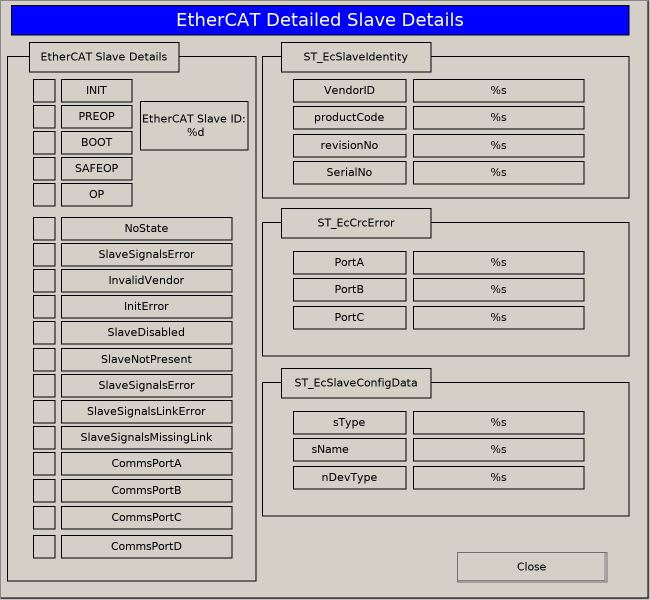
VISUALIZATION diagEtherCATSlaveDetail  // 650x600
VAR_IN_OUT
	//DetailedDataValues:typeEtherCATIndicator;
END_VAR
    Rectangle (0,0 648x598)
    Rectangle (262,56 367x142)
    Rectangle (7,56 249x525)
    Rectangle (33,79 22x23), colour toggle: etherCATdiag.detailDiag.currentState.state = EtherCATstate.INIT
    Rectangle (61,79 71x23), "INIT"
    Rectangle (33,105 22x23), colour toggle: etherCATdiag.detailDiag.currentState.state = EtherCATstate.PREOP
    Rectangle (61,105 71x23), "PREOP"
    Rectangle (33,131 22x23), colour toggle: etherCATdiag.detailDiag.currentState.state = EtherCATstate.BOOT
    Rectangle (61,131 71x23), "BOOT"
    Rectangle (33,157 22x23), colour toggle: etherCATdiag.detailDiag.currentState.state = EtherCATstate.SAFEOP
    Rectangle (61,157 71x23), "SAFEOP"
    Rectangle (33,183 22x23), colour toggle: etherCATdiag.detailDiag.currentState.state = EtherCATstate.OP
    Rectangle (61,183 71x23), "OP"
    Rectangle (33,217 22x23), colour toggle: etherCATdiag.detailDiag.currentState.suffix = EtherCATSuffix.NoState
    Rectangle (61,217 171x23), "NoState"
    Rectangle (33,243 22x23), colour toggle: etherCATdiag.detailDiag.currentState.suffix = EtherCATSuffix.SlaveSignalsError
    Rectangle (61,243 171x23), "SlaveSignalsError"
    Rectangle (33,269 22x23), colour toggle: etherCATdiag.detailDiag.currentState.suffix = EtherCATSuffix.InvalidVendor
    Rectangle (61,269 171x23), "InvalidVendor"
    Rectangle (33,295 22x23), colour toggle: etherCATdiag.detailDiag.currentState.suffix = EtherCATSuffix.InitError
    Rectangle (61,295 171x23), "InitError"
    Rectangle (33,321 22x23), colour toggle: etherCATdiag.detailDiag.currentState.suffix = EtherCATSuffix.SlaveDisabled
    Rectangle (61,321 171x23), "SlaveDisabled"
    Rectangle (33,348 22x23), colour toggle: etherCATdiag.detailDiag.currentState.suffix = EtherCATSuffix.SlaveNotPresent
    Rectangle (61,348 171x23), "SlaveNotPresent"
    Rectangle (33,374 22x23), colour toggle: etherCATdiag.detailDiag.currentState.suffix = EtherCATSuffix.SlaveSignalsError
    Rectangle (61,374 171x23), "SlaveSignalsError"
    Rectangle (33,400 22x23), colour toggle: etherCATdiag.detailDiag.currentState.suffix = EtherCATSuffix.SlaveSignalsLinkError
    Rectangle (61,400 171x23), "SlaveSignalsLinkError"
    Rectangle (33,426 22x23), colour toggle: etherCATdiag.detailDiag.currentState.suffix = EtherCATSuffix.SlaveSignalsMissingLink
    Rectangle (61,426 171x23), "SlaveSignalsMissingLink"
    Rectangle (33,452 22x23), colour toggle: etherCATdiag.detailDiag.currentState.suffix = EtherCATSuffix.CommsPortA
    Rectangle (61,452 171x23), "CommsPortA"
    Rectangle (33,479 22x23), colour toggle: etherCATdiag.detailDiag.currentState.suffix = EtherCATSuffix.CommsPortB
    Rectangle (61,479 171x23), "CommsPortB"
    Rectangle (33,506 22x23), colour toggle: etherCATdiag.detailDiag.currentState.suffix = EtherCATSuffix.CommsPortC
    Rectangle (61,506 171x23), "CommsPortC"
    Rectangle (33,535 22x23), colour toggle: etherCATdiag.detailDiag.currentState.suffix = EtherCATSuffix.CommsPortD
    Rectangle (61,535 171x23), "CommsPortD"
    Rectangle (29,42 150x30), "EtherCAT Slave Details"
    Rectangle (293,79 113x23), "VendorID"
    Rectangle (413,79 171x23), "%s", text variable: etherCATdiag.detailDiag.ConfigData.stSlaveIdentity.vendorId
    Rectangle (413,106 171x23), "%s", text variable: etherCATdiag.detailDiag.ConfigData.stSlaveIdentity.productCode
    Rectangle (293,106 113x23), "productCode"
    Rectangle (293,134 113x23), "revisionNo"
    Rectangle (413,134 171x23), "%s", text variable: etherCATdiag.detailDiag.ConfigData.stSlaveIdentity.revisionNo
    Rectangle (413,161 171x23), "%s", text variable: etherCATdiag.detailDiag.ConfigData.stSlaveIdentity.serialNo
    Rectangle (293,161 113x23), "SerialNo"
    Rectangle (281,42 150x30), "ST_EcSlaveIdentity"
    Rectangle (262,222 367x134)
    Rectangle (293,251 113x23), "PortA"
    Rectangle (413,251 171x23), "%s", text variable: etherCATdiag.detailDiag.crcCount.portA
    Rectangle (413,278 171x23), "%s", text variable: etherCATdiag.detailDiag.crcCount.portB
    Rectangle (293,278 113x23), "PortB"
    Rectangle (293,306 113x23), "PortC"
    Rectangle (413,306 171x23), "%s", text variable: etherCATdiag.detailDiag.crcCount.portC
    Rectangle (281,208 150x30), "ST_EcCrcError"
    Rectangle (262,382 367x134)
    Rectangle (293,411 113x23), "sType"
    Rectangle (413,411 171x23), "%s", text variable: etherCATdiag.detailDiag.ConfigData.sType
    Rectangle (413,438 171x23), "%s", text variable: etherCATdiag.detailDiag.ConfigData.sName
    Rectangle (293,438 113x23), "sName"
    Rectangle (293,466 113x23), "nDevType"
    Rectangle (413,466 171x23), "%s", text variable: etherCATdiag.detailDiag.ConfigData.nDevType
    Rectangle (281,368 150x30), "ST_EcSlaveConfigData"
    Button (457,552 150x30), "Close"
        OnMouseClick: CloseDialog Dialog=diagEtherCATSlaveDetail, Result=OK, NumpadKeypadSet=True
    Rectangle (11,5 618x30), "EtherCAT Detailed Slave Details"
    Rectangle (140,101 108x49), "EtherCAT Slave ID: %d", text variable: etherCATdiag.detailDiagNum
END_VISUALIZATION

(* stored: Version 1.1.0.1, ProductVersion 3.1.4024.12
   Visu diagEtherCATSlaveDetail: Id {0e5479e1-51c5-4cc7-a392-006154e867e5} *)
